FUNCTION_BLOCK TestFB1DeviceSubdevice
VAR_INPUT
END_VAR
VAR_OUTPUT
END_VAR
VAR
	NonPerstInt1:INT:=9;
	NonPerstInt2:INT:=10;
END_VAR
VAR PERSISTENT
	PersInt1:INT:=435;
END_VAR

PersInt1:=PersInt1+1;

END_FUNCTION_BLOCK

(* stored: Version 1.1.0.1, ProductVersion 3.1.4024.6
   POU TestFB1DeviceSubdevice: Id {0cf00b96-6a2b-4955-8ad2-9f608065162c}, SpecialFunc None *)
